FUNCTION_BLOCK CentralController (* Basic Function Block Type *)
  (* Standard: 61499-2 *)
  (* Version 0.0, 1/14/2024, midxav, Template *)
  PACKAGE Main;
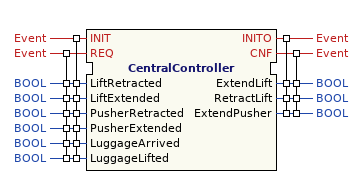
  EVENT_INPUT
    INIT WITH LiftRetracted, LiftExtended, PusherRetracted, PusherExtended, LuggageArrived, LuggageLifted; (* Initialization Request *)
    REQ WITH LiftRetracted, LiftExtended, PusherRetracted, PusherExtended, LuggageArrived, LuggageLifted; (* Normal Execution Request *)
  END_EVENT
  EVENT_OUTPUT
    INITO WITH ExtendLift, RetractLift, ExtendPusher; (* Initialization Confirm *)
    CNF WITH ExtendLift, RetractLift, ExtendPusher; (* Execution Confirmation *)
  END_EVENT
  VAR_INPUT
    LiftRetracted : BOOL; (* Input event qualifier *)
    LiftExtended : BOOL;
    PusherRetracted : BOOL;
    PusherExtended : BOOL;
    LuggageArrived : BOOL;
    LuggageLifted : BOOL;
  END_VAR
  VAR_OUTPUT
    ExtendLift : BOOL; (* Output event qualifier *)
    RetractLift : BOOL;
    ExtendPusher : BOOL;
  END_VAR
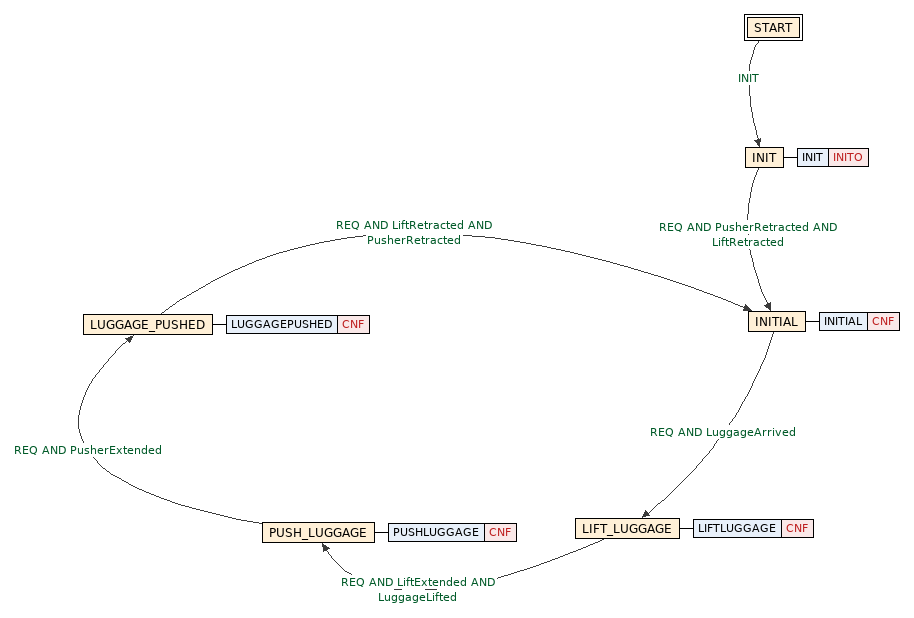
  EC_STATES
    START; (* Initial State *)
    INIT : INIT -> INITO; (* Initialization *)
    INITIAL : INITIAL -> CNF;
    LIFT_LUGGAGE : LIFTLUGGAGE -> CNF;
    PUSH_LUGGAGE : PUSHLUGGAGE -> CNF;
    LUGGAGE_PUSHED : LUGGAGEPUSHED -> CNF;
  END_STATES
  EC_TRANSITIONS
    START TO INIT := INIT;
    INIT TO INITIAL := REQ AND PusherRetracted AND LiftRetracted;
    INITIAL TO LIFT_LUGGAGE := REQ AND LuggageArrived;
    LIFT_LUGGAGE TO PUSH_LUGGAGE := REQ AND LiftExtended AND LuggageLifted;
    PUSH_LUGGAGE TO LUGGAGE_PUSHED := REQ AND PusherExtended;
    LUGGAGE_PUSHED TO INITIAL := REQ AND LiftRetracted AND PusherRetracted;
  END_TRANSITIONS
  ALGORITHM INIT IN ST: (* Initialization algorithm *)
ExtendPusher:= FALSE;
ExtendLift:= FALSE;
RetractLift:=TRUE;
  END_ALGORITHM
  ALGORITHM INITIAL IN ST:
RetractLift:=FALSE;
  END_ALGORITHM
  ALGORITHM LIFTLUGGAGE IN ST:
ExtendLift:=TRUE;
  END_ALGORITHM
  ALGORITHM PUSHLUGGAGE IN ST:
ExtendPusher:=TRUE;
ExtendLift:=FALSE;
  END_ALGORITHM
  ALGORITHM LUGGAGEPUSHED IN ST:
RetractLift:=TRUE;
ExtendPusher:=FALSE;
  END_ALGORITHM
END_FUNCTION_BLOCK
